// TIA Portal V19 export
VAR_GLOBAL   // PLC tag table "NEW OUTPUTS"
   "MFG FEED PUMP OP" AT %Q0.0 : Bool;
   "RO 1 HPP PUMP OP" AT %Q0.1 : Bool;
   "RO 2 HPP PUMP OP" AT %Q0.2 : Bool;
   "CIP PUMP OP" AT %Q0.3 : Bool;
   "PW TRANSFER PUMP W OP" AT %Q0.4 : Bool;
   "PW TRANSFER PUMP S OP" AT %Q0.5 : Bool;
   "SPARE OP1" AT %Q0.6 : Bool;
   "SPARE OP2" AT %Q0.7 : Bool;
   "SPARE OP3" AT %Q1.0 : Bool;
   "DP-1 OP" AT %Q1.1 : Bool;
   "DP-2 OP" AT %Q12.0 : Bool;
   "UV-1 OP" AT %Q12.1 : Bool;
   "SPARE OP4" AT %Q12.2 : Bool;
   "SPARE OP5" AT %Q12.3 : Bool;
   "SPARE OP6" AT %Q12.4 : Bool;
   "SPARE OP7" AT %Q12.5 : Bool;
   "SPARE OP8" AT %Q12.6 : Bool;
   "HOOTER OP" AT %Q12.7 : Bool;
   "MFG OPEN V1" AT %Q13.0 : Bool;
   "MFG OPEN V2" AT %Q13.2 : Bool;
   "MFG OPEN V3" AT %Q13.4 : Bool;
   "MFG OPEN V4" AT %Q13.6 : Bool;
   "MFG OPEN V5" AT %Q16.0 : Bool;
   "MFG CLOSE V1" AT %Q13.1 : Bool;
   "MFG CLOSE V2" AT %Q13.3 : Bool;
   "MFG CLOSE V3" AT %Q13.5 : Bool;
   "MFG CLOSE V4" AT %Q13.7 : Bool;
   "MFG CLOSE V5" AT %Q16.1 : Bool;
   "ACF OPEN V1" AT %Q16.2 : Bool;
   "ACF OPEN V2" AT %Q16.4 : Bool;
   "ACF OPEN V3" AT %Q16.6 : Bool;
   "ACF OPEN V4" AT %Q17.0 : Bool;
   "ACF OPEN V5" AT %Q17.2 : Bool;
   "ACF CLOSE V1" AT %Q16.3 : Bool;
   "ACF CLOSE V2" AT %Q16.5 : Bool;
   "ACF CLOSE V3" AT %Q16.7 : Bool;
   "ACF CLOSE V4" AT %Q17.1 : Bool;
   "ACF CLOSE V5" AT %Q17.3 : Bool;
   "SF OPEN V1" AT %Q17.4 : Bool;
   "SF OPEN V2" AT %Q17.6 : Bool;
   "SF OPEN V3" AT %Q20.0 : Bool;
   "SF OPEN V4" AT %Q20.2 : Bool;
   "SF OPEN V5" AT %Q20.4 : Bool;
   "SF OPEN V6" AT %Q20.6 : Bool;
   "SF OPEN V7" AT %Q21.0 : Bool;
   "SF CLOSE V1" AT %Q17.5 : Bool;
   "SF CLOSE V2" AT %Q17.7 : Bool;
   "SF CLOSE V3" AT %Q20.1 : Bool;
   "SF CLOSE V4" AT %Q20.3 : Bool;
   "SF CLOSE V5" AT %Q20.5 : Bool;
   "SF CLOSE V6" AT %Q20.7 : Bool;
   "SF CLOSE V7" AT %Q21.1 : Bool;
   "AV 1" AT %Q21.2 : Bool;
   "AV 2" AT %Q21.3 : Bool;
   "AV 3" AT %Q21.4 : Bool;
   "AV 4" AT %Q21.5 : Bool;
   "SPARE OP9" AT %Q21.6 : Bool;
   "SPARE OP10" AT %Q21.7 : Bool;
END_VAR
